// TIA Portal project "giris_bitini_takip_etme" (V18)

(* hardware
DEVICE "S7-1200 station_1"  S7-1200 Station
   slot 0: "Rack_0"  S7-1200 Rack  Rack  V1.0
   slot 1: "PLC_1"  CPU 1214C AC/DC/Rly  6ES7 214-1BG40-0XB0  V4.6
*)

// ===== PLC "PLC_1"  CPU 1214C AC/DC/Rly =====

VAR_GLOBAL   // PLC tag table "Default tag table"
   "Tag_1" AT %IB0 : Byte;
   "Tag_2" AT %MD0 : DWord;
   "Tag_3" AT %MD4 : DWord;
   "Tag_4" AT %MD30 : DWord;
   "Tag_5" AT %MD50 : UDInt;
END_VAR

ORGANIZATION_BLOCK "Main"   // OB1, LAD, ProgramCycle
TITLE = "Main Program Sweep (Cycle)"
{ S7_Optimized_Access := 'TRUE' }
VERSION : 0.1
   VAR_INPUT
      Initial_Call : Bool;   // Initial call of this OB
      Remanence : Bool;   // =True, if remanent data are available
   END_VAR
BEGIN

REGION Network 1
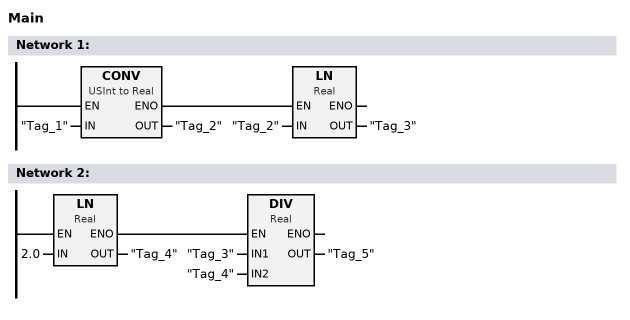
   "Tag_2" := USINT_TO_REAL("Tag_1");
   "Tag_3" := LN("Tag_2");
END_REGION

REGION Network 2
   "Tag_4" := LN(2.0);
   "Tag_5" := "Tag_3" / "Tag_4";
END_REGION
END_ORGANIZATION_BLOCK